FUNCTION_BLOCK FB_PositionState_Defaults
VAR_IN_OUT
    stPositionState: DUT_PositionState;
END_VAR
VAR_INPUT
    fVeloDefault: LREAL;
    fDeltaDefault: LREAL;
    fAccelDefault: LREAL;
    fDecelDefault: LREAL;
END_VAR

IF stPositionState.fVelocity = 0 THEN
    stPositionState.fVelocity := fVeloDefault;
END_IF
IF stPositionState.fDelta = 0 THEN
    stPositionState.fDelta := fDeltaDefault;
END_IF
IF stPositionState.fAccel = 0 THEN
    stPositionState.fAccel := fAccelDefault;
END_IF
IF stPositionState.fDecel = 0 THEN
    stPositionState.fDecel := fDecelDefault;
END_IF

END_FUNCTION_BLOCK

(* stored: Version 1.1.0.1, ProductVersion 3.1.4022.18
   POU FB_PositionState_Defaults: Id {5f326ffa-3869-4f51-b9bc-bdf476cd3f65}, SpecialFunc None *)
